TYPE E_ArrayOrder :
(
	RowWiseSaw,
	RowWiseMeander,
	ColWiseSaw,
	ColWiseMeander
)USINT;
END_TYPE

(* stored: Version 1.1.0.1, ProductVersion 3.1.0.25
   DUT E_ArrayOrder: Id {3e8ad601-f223-482a-b74f-4325821be8a2} *)
